{attribute 'TcGenerated'}
{attribute 'no-analysis'}
{attribute 'linkalways'}
// This function has been automatically generated from the project information.
VAR_GLOBAL CONSTANT
	{attribute 'const_non_replaced'}
	stLibVersion_BaseClassExampleProgram : ST_LibVersion := (iMajor := 1, iMinor := 1, iBuild := 15, iRevision := 0, nFlags := 0, sVersion := '1.1.15.0');
END_VAR

(* stored: Version 1.1.0.1, ProductVersion 3.1.4024.9
   GVL Global_Version: Id {73cae4cc-7ad5-4a8c-b591-f94f84666b18} *)
